Staubli VAL3: onF1Event.pgx

program onF1Event()
begin
  // look if the bButton is enable
  if bButton[0]
    //
  endIf
end
